INTERFACE ITF_CANControl

METHOD M_GetMessage : BOOL
VAR_INPUT
END_VAR
END_METHOD

METHOD M_PushMessage : BOOL
VAR_INPUT
	messageSend : ST_TxRxMessage;
END_VAR
END_METHOD

END_INTERFACE

(* stored: Version 1.1.0.1, ProductVersion 3.1.4024.9
   Itf ITF_CANControl: Id {3cc4a4bf-782b-4cdf-9b13-ee48a44f9498}
   Method M_GetMessage: Id {b1e1187f-ac09-4b80-8a54-9f02690a542a}
   Method M_PushMessage: Id {654feaee-b537-49f8-b74e-8496d9a78cf2} *)
